// TwinCAT 3 PLC project Untitled1
// ProgramVersion: 3.1.4024.0
// libraries:
//   Tc2_Standard, * (Beckhoff Automation GmbH)
//   Tc2_System, * (Beckhoff Automation GmbH)
//   Tc3_Module, * (Beckhoff Automation GmbH)
// project tree:
//   DUTs/ E_ProductType.TcDUT, ST_ProductInfo.TcDUT
//   / PlcTask.TcTTO
//   POUs/ FB_Blokgolf.TcPOU, FB_Inventory.TcPOU, MAIN.TcPOU, F_Calc.TcPOU
// real-time tasks:
//   TASK PlcTask: cycle T#1ms, priority 20, ADS port 350

CONFIGURATION Untitled1
    RESOURCE PLC ON TwinCAT3
        TASK PlcTask(INTERVAL := T#1ms, PRIORITY := 20);
        PROGRAM MAIN WITH PlcTask : MAIN;
    END_RESOURCE
END_CONFIGURATION

// ---- DUTs/E_ProductType.TcDUT
{attribute 'qualified_only'}
{attribute 'strict'}
TYPE E_ProductType:
(
	cube,
	cylinder,
	sphere			
)
;
END_TYPE

// ---- DUTs/ST_ProductInfo.TcDUT
TYPE ST_ProductInfo :
STRUCT
	eproductType:	E_ProductType;
	fSpecificWeight: REAL;
	fDimension1 : REAL;
	fDimension2 : REAL;
	fDimension3 : REAL;
END_STRUCT
END_TYPE

// ---- POUs/MAIN.TcPOU
PROGRAM MAIN
VAR
	//blockgolf1: FB_Blokgolf;
	_product1: ST_ProductInfo := (eproductType := E_ProductType.cube, fDimension1 := 10, fDimension2 := 5, fDimension3 := 12, fSpecificWeight := 1000);
	_product2: ST_ProductInfo := (eproductType := E_ProductType.cylinder, fDimension1 := 20, fDimension2 := 10, fDimension3 := 24, fSpecificWeight := 2000);
	inventory1: FB_Inventory(product1 := _product1, product2 := _product2);
	bTest: BOOL;

END_VAR

IF bTest THEN
	inventory1.M_Add(_product2);
	inventory1.M_Remove(0);
	bTest := FALSE;
END_IF

END_PROGRAM

// ---- POUs/FB_Inventory.TcPOU
FUNCTION_BLOCK FB_Inventory
VAR_INPUT
END_VAR
VAR_OUTPUT
END_VAR
VAR
	_stInventory : ARRAY [0..5] OF ST_ProductInfo;
	_nNumberProducts : INT := 0;
	_fTotalWeight : REAL;
	_fTotalVolume : REAL;
END_VAR

METHOD FB_init : BOOL
VAR_INPUT
	bInitRetains : BOOL; // if TRUE, the retain variables are initialized (warm start / cold start)
	bInCopyCode : BOOL;  // if TRUE, the instance afterwards gets moved into the copy code (online change)
	product1 : ST_ProductInfo;
	product2 : ST_ProductInfo;
END_VAR
M_Add(product1);
M_Add(product2);
END_METHOD

PROPERTY PUBLIC fTotalVolume : REAL
GET
END_GET
SET
END_SET
END_PROPERTY

PROPERTY PUBLIC fTotalWeight : REAL
GET
END_GET
SET
END_SET
END_PROPERTY

METHOD PUBLIC M_Add
VAR_INPUT
	stProductInfo : ST_ProductInfo;
END_VAR
_stInventory[_nNumberProducts] := stProductInfo;
_nNumberProducts := _nNumberProducts + 1;
END_METHOD

METHOD PRIVATE M_CalculateVolume
VAR_INPUT
END_VAR
END_METHOD

METHOD PRIVATE M_CalculateWeight
VAR_INPUT
END_VAR
END_METHOD

METHOD PUBLIC M_Remove
VAR_INPUT
	nIndex : INT;
END_VAR
VAR
	stNullProduct : ST_ProductInfo := (eproductType := E_ProductType.cube, fDimension1 := 0, fDimension2 := 0, fDimension3 := 0, fSpecificWeight := 0);
END_VAR
_stInventory[nIndex] := _stInventory[_nNumberProducts - 1];
_stInventory[_nNumberProducts - 1] := stNullProduct;
_nNumberProducts := _nNumberProducts - 1;
END_METHOD

PROPERTY PUBLIC nNumberProducts : INT
GET
END_GET
SET
END_SET
END_PROPERTY

PROPERTY PUBLIC stInventory : array [1..5] of ST_ProductInfo
GET
END_GET
SET
END_SET
END_PROPERTY

END_FUNCTION_BLOCK

// ---- POUs/FB_Blokgolf.TcPOU
FUNCTION_BLOCK FB_Blokgolf
VAR_INPUT
END_VAR
VAR_OUTPUT
END_VAR
VAR
	_timer1 : TP;
	_timer2 : TP;
	bEnabled: BOOL;
END_VAR

_timer1.IN := bEnabled AND NOT _timer2.Q;
_timer1();

_timer2.IN := bEnabled AND NOT _timer1.Q;
_timer2();

PROPERTY PUBLIC bSignalOut : BOOL
GET
END_GET
SET
END_SET
END_PROPERTY

METHOD PUBLIC M_Start
VAR_INPUT
	onTime : TIME;
	offTime : TIME;
END_VAR
bEnabled := TRUE;
_timer1.PT := onTime;
_timer2.PT := offTime;
END_METHOD

METHOD PUBLIC M_Stop
VAR_INPUT
END_VAR
bEnabled := false;
END_METHOD

PROPERTY PUBLIC nCounter : REAL
GET
END_GET
SET
END_SET
END_PROPERTY

END_FUNCTION_BLOCK

// ---- POUs/F_Calc.TcPOU
FUNCTION_BLOCK F_Calc
VAR_INPUT
	nGetal : INT := 0;
END_VAR
VAR_OUTPUT
	
END_VAR
VAR
	_fAns : REAL;
	_fSavedValue : REAL;
END_VAR

PROPERTY PUBLIC fAns : REAL
GET
fAns := _fAns;
END_GET
END_PROPERTY

PROPERTY PUBLIC fSavedValue : REAL
GET
fSavedValue := _fSavedValue;
END_GET
SET
VAR
	//fGetal : REAL;
END_VAR
_fSavedValue := fSavedValue;
END_SET
END_PROPERTY

METHOD PUBLIC M_Add : REAL
VAR_INPUT
		getalOmOpTeTellen : REAL ;
END_VAR
_fAns := _fAns + getalOmOpTeTellen;
END_METHOD

METHOD PUBLIC M_Divide : REAL
VAR_INPUT
		GetalOmTeDelen : REAL;
END_VAR
_fAns := _fAns / GetalOmTeDelen;
END_METHOD

METHOD PUBLIC M_Multiply : REAL
VAR_INPUT
	GetalOmTeVermenigvuldigen : REAL;
END_VAR
_fAns := _fAns * GetalOmTeVermenigvuldigen;
END_METHOD

METHOD PUBLIC M_Save
VAR_INPUT
END_VAR
_fSavedValue := _fAns;
END_METHOD

METHOD PUBLIC M_Subtract : REAL
VAR_INPUT
	getalOmAfTeTrekken : REAL;
END_VAR
_fAns := _fAns - getalOmAfTeTrekken;
END_METHOD

END_FUNCTION_BLOCK
